// LS Electric XG5000 project: 2차 프로젝트 컨베이어 제어 코드(모드버스 RTU서버 버전)
// PLC LSPLC
// module base 0 slot 0: 입출력 모듈:XBC-DR32H (DC 24V 입력, 릴레이 출력 32점)

PROGRAM NewProgram (task: 스캔 프로그램)

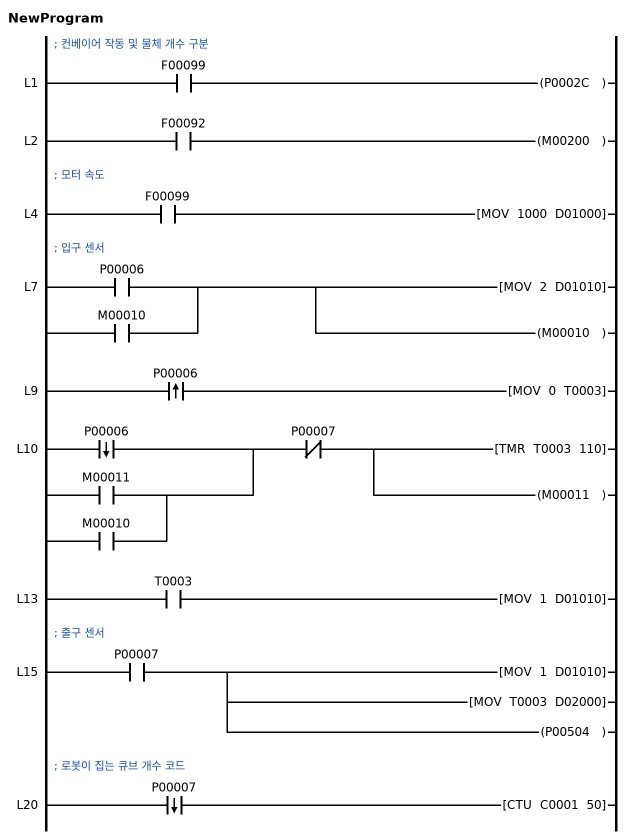
// 컨베이어 작동 및 물체 개수 구분
; L1
LOAD      F00099
OUT       P0002C
; L2
LOAD      F00092
OUT       M00200
// 모터 속도
; L4
LOAD      F00099
MOV       1000 D01000
// 입구 센서
; L7
LOAD      P00006
OR        M00010
MOV       2 D01010
OUT       M00010
; L9
LOADP     P00006
MOV       0 T0003
; L10
LOADN     P00006
OR        M00011
OR        M00010
AND NOT   P00007
TMR       T0003 110
OUT       M00011
; L13
LOAD      T0003
MOV       1 D01010
// 출구 센서
; L15
LOAD      P00007
MOV       1 D01010
MOV       T0003 D02000
OUT       P00504
// 로봇이 집는 큐브 개수 코드
; L20
LOADN     P00007
CTU       C0001 50